Universal Robots PolyScope program: measure_fluffiness.urp

Program measure_fluffiness (installation=default directory=/programs/Nicolas_Arteaga createdIn=5.12.6.1102099 lastSavedIn=5.12.4.1101661 robotSerialNumber=20225502378)
Calibrated DH parameters: a=[0.00022, -0.425328, -0.389701, 0.000059, 0.000065, 0]; d=[0.162608, 0.803456, 9.992211, -10.662202, 0.099702, 0.099559]; alpha=[1.570756, 0.001543, 0.004316, 1.570651, -1.570122, 0]; deltaTheta=[0, 0.002917, 0.116094, -0.119008, 0, -0.000001]
Robot Program (runOnlyOnce=true)
  MoveJ speed 60 deg/s, acceleration 80 deg/s^2 (useActiveTCP=true) feature=Base
    Waypoint Waypoint_1: TCP in base x=227.087 y=826.923 z=352.054 mm, rx=-1.5343 ry=-1.0982 rz=-1.6415 rad; joints [-112.615, -64.832, 77.78, -11.56, 94.974, 81.449] deg; TCP offset x=0 y=0 z=191.5 mm, rx=0 ry=0 rz=0 rad
    URCap Gripper Activate (Robotiq_Grippers, Robotiq Inc.) dataModel(ResetAndActivateKey=false)
    URCap Gripper (Robotiq_Grippers, Robotiq Inc.) dataModel(position=100.0, force=100.0, speed=50.0, positionInDouble=100.0, forceInDouble=100.0, speedInDouble=50.0, slaveIds=[9], blocking=true)
    MoveJ speed 60 deg/s, acceleration 80 deg/s^2 (useActiveTCP=true) feature=Base
      Waypoint Waypoint_2: TCP in base x=227.112 y=826.899 z=142.725 mm, rx=-1.5343 ry=-1.0982 rz=-1.6415 rad; joints [-112.624, -52.3, 91.664, -37.98, 95.052, 81.42] deg
      Waypoint Waypoint_1: TCP in base x=227.087 y=826.923 z=352.054 mm, rx=-1.5343 ry=-1.0982 rz=-1.6415 rad; joints [-112.615, -64.832, 77.78, -11.56, 94.974, 81.449] deg
      URCap Gripper (Robotiq_Grippers, Robotiq Inc.) dataModel(position=83.0, force=100.0, speed=100.0, positionInDouble=83.0, forceInDouble=100.0, speedInDouble=100.0, slaveIds=[9], blocking=true)
